PROGRAM Axis03_Status
VAR
	Always_ON	:	BOOL	:=TRUE	;//상시 ON 
	Always_OFF	:	BOOL	:=FALSE	;//상시 OFF
END_VAR

// NETWORK 1

END_PROGRAM

(* stored: Version 1.1.0.1, ProductVersion 3.1.4024.15
   POU Axis03_Status: Id {6772cf1a-0606-4815-9c2e-28638ae5dcce}, SpecialFunc None *)
